// TIA Portal V21 export
DATA_BLOCK "12312"   // DB2
{ S7_Optimized_Access := 'TRUE' }
   VAR
      wad : Real;
      xawd : Bool;
   END_VAR
BEGIN
END_DATA_BLOCK
